FUNCTION_BLOCK ZONA

VAR_INPUT
	ENABLE     : BOOL;
	RIPRISTINO : BOOL;
	LIBERO_I   : BOOL;
	TRIGGER_I  : BOOL;
END_VAR

VAR_OUTPUT
	LIBERO_O   : BOOL;
	TRIGGER_O  : BOOL;
END_VAR

VAR
END_VAR

END_FUNCTION_BLOCK

(* stored: Version 1.1.0.1, ProductVersion 3.1.4024.12
   POU ZONA: Id {90ca5c29-741d-449a-91f5-50a6a2a13047}, SpecialFunc None *)
